(*
SPDX-FileCopyrightText: © 2026 Oleksandr Tiutyk <trofimich@gmail.com>
SPDX-License-Identifier: MIT
License: https://opensource.org/license/mit
*)

(*!
<summary>Reports an argument value outside the range accepted by the caller.</summary>
<description>
The caller determines that the argument is invalid; Throw formats the diagnostic rather than validating the
argument. Argument values are represented in at most 255 characters. STRING and WSTRING values longer than 255
characters retain their first 254 characters followed by an ellipsis. Dynamic exceptions belong to the current
task memory manager until cleanup.
</description>
*)
INTERFACE IArgumentOutOfRangeException EXTENDS IGeneralException

(*!
<summary>Formats the rejected argument and propagates the exception with source metadata.</summary>
<description>
Call in the owning cyclic task, not during FB_init. Reads the supplied value only during this call and retains
its formatted text. Long STRING and WSTRING values use a 254-character prefix followed by an ellipsis; exactly
255 characters are kept unchanged. Other types use the shared ANY formatter. Sets error code to zero and has
no inner cause. Builder or exception allocation failure uses the terminal memory mechanism.
</description>
<param name="argumentName">Name of the argument rejected by the caller.</param>
<param name="argumentValue">Live value to describe; string inputs must be null-terminated.</param>
*)
METHOD Throw
VAR_INPUT
	sourceNamespaceName : STRING;
	sourceClassName : STRING;
	sourcePOUName : STRING;
	sourcePosition : STRING;
	argumentName : STRING;
	argumentValue : ANY;
END_VAR
END_METHOD

END_INTERFACE

(* stored: Version 1.1.0.1
   Itf IArgumentOutOfRangeException: Id {b593408e-8234-4422-a350-6b47381deafa}
   Method Throw: Id {3a3b6fab-8c6a-43b0-a149-d2423f42faeb} *)
